FUNCTION_BLOCK PUBLIC FB_SubjectBase IMPLEMENTS I_Subject
VAR
	aObservers			: ARRAY [1..Param.cMaxObservers] OF I_Observer;
END_VAR

METHOD PUBLIC Attach : BOOL
VAR_INPUT
	ipObserver				: I_Observer;
END_VAR
VAR
	nIndex					: INT := 0;
END_VAR
Attach := FALSE;
IF (ipObserver = 0) THEN
	RETURN;
END_IF

// is the observer already registered?
FOR nIndex := 1 TO Param.cMaxObservers DO	
	IF (THIS^.aObservers[nIndex] = ipObserver) THEN
		RETURN;
	END_IF
END_FOR

// save the observer object into the array of observers and send the actual value
FOR nIndex := 1 TO Param.cMaxObservers DO
	IF (THIS^.aObservers[nIndex] = 0) THEN
		THIS^.aObservers[nIndex] := ipObserver;
		Attach := TRUE;
		EXIT;					
	END_IF
END_FOR
END_METHOD

METHOD PUBLIC Detach : BOOL
VAR_INPUT
	ipObserver		: I_Observer;
END_VAR
VAR
	nIndex			: INT := 0;
END_VAR
Detach := FALSE;
IF (ipObserver = 0) THEN
	RETURN;
END_IF

FOR nIndex := 1 TO Param.cMaxObservers DO
	IF (THIS^.aObservers[nIndex] = ipObserver) THEN
		THIS^.aObservers[nIndex] := 0;
		Detach := TRUE;	
	END_IF
END_FOR
END_METHOD

END_FUNCTION_BLOCK

(* stored: Version 1.1.0.1, ProductVersion 3.1.4022.10
   POU FB_SubjectBase: Id {1555c4fa-9f19-4104-9eaa-bc0df5e50c20}, SpecialFunc None
   Method Attach: Id {f06878e3-4aca-4636-a252-4cd39b77b47d}
   Method Detach: Id {2c62a29a-ed94-4578-afe6-e2c2a1804903} *)
